// Gets the lower bound index of the array of specified type.
FUNCTION F_GetWStringArrayLowerBound : T_Position // The lower bound index of the specified array.
VAR_IN_OUT
	arArray : ARRAY[*] OF WSTRING; // The array to query.
END_VAR

F_GetWStringArrayLowerBound := LOWER_BOUND(arArray, 1);

END_FUNCTION

(* stored: Version 1.1.0.1
   POU F_GetWStringArrayLowerBound: Id {a95c65b5-6b09-048c-2911-2880746a98e9}, SpecialFunc None *)
